FUNCTION_BLOCK FB_FT_PT1 (* low pass filter with a programmable time T and faktor K *)
  (* Standard: OSCAT; Classification: Control *)
  (* Version 0.0, 2011-06-21, 4DIAC-IDE, 4DIAC-Consortium *)
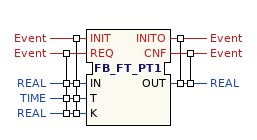
  EVENT_INPUT
    INIT WITH IN, T, K; (* Initialization Request *)
    REQ WITH IN, T, K; (* Normal Execution Request *)
  END_EVENT
  EVENT_OUTPUT
    INITO WITH OUT; (* Initialization Confirm *)
    CNF WITH OUT; (* Execution Confirmation *)
  END_EVENT
  VAR_INPUT
    IN : REAL; (* Input signal *)
    T : TIME := 1.0; (* Time constant *)
    K : REAL := 1.0; (* Amplification factor *)
  END_VAR
  VAR_OUTPUT
    OUT : REAL; (* Output signal *)
  END_VAR
  VAR
    tx : DWORD; (* actual time *)
    last : DWORD; (* last time *)
  END_VAR
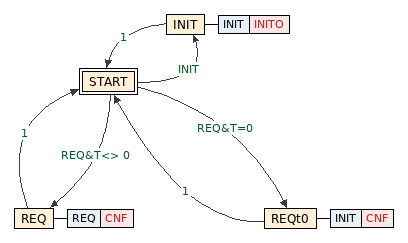
  EC_STATES
    START; (* Initial State *)
    INIT : INIT -> INITO; (* Initialization *)
    REQ : REQ -> CNF; (* Normal execution *)
    REQt0 : INIT -> CNF;
  END_STATES
  EC_TRANSITIONS
    START TO INIT := INIT;
    INIT TO START := 1;
    REQ TO START := 1;
    START TO REQ := REQ&T<> 0;
    START TO REQt0 := REQ&T=0;
    REQt0 TO START := 1;
  END_TRANSITIONS
  ALGORITHM REQ IN AnyText: (* Normally executed algorithm *)
tx() = T_PLC_US();
OUT() = OUT() + (IN() * K() - OUT()) * DWORD_TO_REAL(tx() - last()) / (TIME_TO_REAL(T()) * 1.0E6f);
last() = tx();
  END_ALGORITHM
  ALGORITHM INIT IN AnyText: (* Initialization algorithm *)
tx() = T_PLC_US();
OUT() = K() * IN();
last() = tx();
  END_ALGORITHM
END_FUNCTION_BLOCK
